(* IEC 61131-3 sources: volt/packages/volt-lsp-iec/test-corpus/pro2193/Device/Plc Logic/Application/99 Library/Function Blocks/Timers, 6 files *)

(* ---- BTOF.pou ---- *)
// Brink-TOF
{attribute 'no_explicit_call' := 'Do not call the body of BTOF directly! Use methods like Set to interact with this FB'}
{attribute 'monitoring_display' := 'TOF1.ET'}
FUNCTION_BLOCK FINAL BTOF
VAR
	TOF1		: Standard.TOF;
END_VAR

// Use methods to interact with the FB.

%LANGUAGE ST

END_FUNCTION_BLOCK

// Reset the timer.
METHOD PUBLIC Reset

%LANGUAGE ST
TOF1(IN := FALSE);

END_METHOD

// Set Brink timer
METHOD PUBLIC Set : BOOL
VAR_INPUT
	In	: BOOL;	// Starts timer with rising edge, stops timer with falling edge
	Pt	: REAL;	// Time to pass (in sec.), before Q is set
END_VAR

%LANGUAGE ST
TOF1(
	IN := In,
	PT := TO_TIME(Pt * 1000),
	Q  => ,
	ET => );

Set := TOF1.Q;

END_METHOD

// Monitor the output Q of the timer
{attribute 'monitoring':='call'}
PROPERTY PUBLIC Q : BOOL

GET
VAR
END_VAR

%LANGUAGE ST
Q := TOF1.Q;

END_GET
END_PROPERTY

(* ---- BTON.pou ---- *)
// Brink-TON
{attribute 'no_explicit_call' := 'Do not call the body of BTOF directly! Use methods like Set to interact with this FB'}
{attribute 'monitoring_display' := 'TON1.ET'}
FUNCTION_BLOCK FINAL BTON
VAR
	TON1		: Standard.TON;
END_VAR

// Use methods to interact with the FB.

%LANGUAGE ST

END_FUNCTION_BLOCK

// Reset the timer.
METHOD PUBLIC Reset

%LANGUAGE ST
TON1(IN := FALSE);

END_METHOD

// Set Brink timer
METHOD PUBLIC Set : BOOL
VAR_INPUT
	In	: BOOL;	// Starts timer with rising edge, stops timer with falling edge
	Pt	: REAL;	// Time to pass (in sec.), before Q is set
END_VAR

%LANGUAGE ST
TON1(
	IN := In,
	PT := TO_TIME(Pt * 1000),
	Q  => ,
	ET => );

Set := TON1.Q;

END_METHOD

// Monitor the output Q of the timer
{attribute 'monitoring':='call'}
PROPERTY PUBLIC Q : BOOL

GET
VAR
END_VAR

%LANGUAGE ST
Q := TON1.Q;

END_GET
END_PROPERTY

(* ---- MeasureTime.pou ---- *)
// Count time (in sec) how long an input is high/active. Counter resets when input is low.
{attribute 'no_explicit_call' := 'Do not call the body of MeasureModuleTime directly! Use methods to interact with this FB'}
{attribute 'hide_all_locals'}
{attribute 'monitoring_display' := 'rStoredTime'}
FUNCTION_BLOCK MeasureTime
VAR_OUTPUT
	rStoredTimeMax	: REAL;
END_VAR
VAR
	TON1			: Standard.TON;
	rStoredTime		: REAL;		// Dynamic - The currently elapsed time while measuring. Resets when a new measurement starts.
END_VAR

%LANGUAGE ST

END_FUNCTION_BLOCK

// Measure the time how long a condition is true.
METHOD PUBLIC Measure : REAL
VAR_INPUT
	In	: BOOL;	// Measure the time the input remains high
END_VAR

%LANGUAGE ST
IF (In XOR TON1.IN)				// Triggers the first cycle In is true, and the first cycle In is false. Give output.
OR (In AND TON1.ET > T#1S)		// Output will start running when timer has been running for more than 1 sec.
THEN
	rStoredTime		:= TO_REAL(TON1.ET) / 1000;
END_IF

IF NOT In AND TON1.IN THEN
	rStoredTimeMax	:= TO_REAL(TON1.ET) / 1000;
END_IF

TON1(
	IN := In,
	PT := GVL_Constants.TimeLongest,
	Q  => ,
	ET => );

Measure := rStoredTime;			// Give the output

END_METHOD

// Get elapsed time value
{attribute 'monitoring':='call'}
PROPERTY PUBLIC ElapsedTime : REAL

GET
VAR
END_VAR

%LANGUAGE ST
ElapsedTime := rStoredTime;

END_GET
END_PROPERTY

(* ---- ONTIME.pou ---- *)
// ONTIME measures the total time that a signal is active
{attribute 'monitoring_display' := 'udiSeconds'}
FUNCTION_BLOCK ONTIME
VAR_INPUT
	In			: BOOL;
END_VAR
VAR
	Last		: CAA.TICK;
	edge		: BOOL;
	udiMs		: UDINT;

	udiSeconds	: UDINT;	// Non-resetting ever-increasing time In is high
	udiCycles	: UDINT;	// Number of times the input switched on
	refSeconds	: REFERENCE TO UDINT REF= udiSeconds;
	refCycles	: REFERENCE TO UDINT REF= udiCycles;
END_VAR

%LANGUAGE ST
Initialize();

IF In THEN
	udiMs			:= udiMs + (TICKU.GetElapsedTimeInUSec(Last) / 1000);	// Add the elapsed milliseconds since last cycle

	IF udiMs >= 1000 THEN		// Check if a second has elapsed
		refSeconds	:= refSeconds + 1;
		udiMs		:= udiMs - 1000;
	END_IF

	refCycles		:= refCycles + TO_UDINT(NOT edge);
END_IF

Last				:= TICKS.GetTick(FALSE);
edge				:= In;

END_FUNCTION_BLOCK

METHOD PRIVATE Initialize
VAR_INST
	{attribute 'init_on_onlchange' }
	xInitialized	: BOOL;
END_VAR

%LANGUAGE ST
IF xInitialized THEN
	RETURN;
END_IF

Last			:= TICKS.GetTick(FALSE);
udiMs			:= 0;

xInitialized	:= TRUE;

END_METHOD

METHOD PUBLIC Reset
VAR_INPUT
END_VAR

%LANGUAGE ST
refSeconds		:= 0;
refCycles		:= 0;

Last			:= TICKS.GetTick(FALSE);
udiMs			:= 0;

END_METHOD

METHOD PUBLIC SetExternalCyclesReference
VAR_INPUT
	Cycles	: REFERENCE TO UDINT;
END_VAR

// We often need to persist the ONTIME data, so the data retains their value after reboots.
// For example if we count how long a vacuumpump has been running.
// In that case we need to declare the data in the PersistentVars list
// Use this method to set a reference to that variable

// If this method is never used (or reference is set to NULL), data is counted internally in the FB.

%LANGUAGE ST
IF __ISVALIDREF(Cycles) THEN
	THIS^.refCycles		REF= Cycles;
ELSE
	THIS^.refCycles		REF= udiCycles;
END_IF

END_METHOD

METHOD PUBLIC SetExternalSecondsReference
VAR_INPUT
	Seconds	: REFERENCE TO UDINT;
END_VAR

// We often need to persist the ONTIME data, so the data retains their value after reboots.
// For example if we count how long a vacuumpump has been running.
// In that case we need to declare the data in the PersistentVars list
// Use this method to set a reference to that variable

// If this method is never used (or reference is set to NULL), data is counted internally in the FB.

%LANGUAGE ST
IF __ISVALIDREF(Seconds) THEN
	THIS^.refSeconds	REF= Seconds;
ELSE
	THIS^.refSeconds	REF= udiSeconds;
END_IF

END_METHOD

{attribute 'monitoring':='call'}
PROPERTY PUBLIC AsReal : REAL

GET
VAR
END_VAR

%LANGUAGE ST
AsReal := TO_REAL(refSeconds) + TO_REAL(udiMs) / 1000;

END_GET
END_PROPERTY

{attribute 'monitoring':='call'}
PROPERTY PUBLIC AsTime : TIME

GET
VAR
END_VAR

%LANGUAGE ST
AsTime := TO_TIME(refSeconds * 1000 + udiMs);

END_GET
END_PROPERTY

{attribute 'monitoring':='call'}
PROPERTY PUBLIC Cycles : ULINT

GET
VAR
END_VAR

%LANGUAGE ST
Cycles := refCycles;

END_GET
END_PROPERTY

{attribute 'monitoring':='call'}
PROPERTY PUBLIC InSeconds : ULINT

GET
VAR
END_VAR

%LANGUAGE ST
InSeconds := refSeconds;

END_GET
END_PROPERTY

(* ---- SignalTimeoutFB.pou ---- *)
// This FB compares the input signal to the expected value, and will throw an alarm when the result is not as expected within a given time.
// The GetValue method returns the input value, and starts the timeout timer.
// The timer runs as long as the GetValue is called in every successive PLC cycle, the first cycle in which it is not called, it will reset the timer.
FUNCTION_BLOCK SignalTimeoutFB
VAR_INPUT
	input		: BOOL;			// Input signal
	timeOut		: REAL := 5;	// Timout for alarm  (default: 5s)
END_VAR
VAR_OUTPUT
	alarmActive	: BOOL;			// Input is not equal to Expected within the given timeout
END_VAR
VAR
	requested	: BOOL;			// Toggle bit for detecting every GetValue call
	timer		: BTON;			// Alarm timer
END_VAR

%LANGUAGE ST
IF NOT requested THEN
	timer.Reset();
	alarmActive := FALSE;
END_IF

requested := FALSE;

END_FUNCTION_BLOCK

// Starts the timeout timer, and returns the input signal
METHOD GetValue : BOOL
VAR_INPUT
	expected : BOOL;
END_VAR

%LANGUAGE ST
alarmActive	:= timer.Set(In := input <> expected, Pt := timeOut);
requested	:= TRUE;
GetValue	:= input;

END_METHOD

(* ---- StopwatchFB.pou ---- *)
// Measure precise durations [µs]. Use to debug code and check how long code needs to run.
// Also use Monitor() method to measure duration of booleans
{attribute 'no_explicit_call' := 'Do not call the body of StopwatchFB directly! Use methods to interact with this FB'}
{attribute 'monitoring_display' := 'actTime'}
{attribute 'symbol' := 'none'}
FUNCTION_BLOCK PUBLIC StopwatchFB
EXTENDS MonitoringAddLogBase
VAR
	ltStart		: LTIME;
END_VAR
VAR_OUTPUT
	actTime		: UDINT;	// UDINT storing microseconds can represent roughly 4,295 seconds or 71,5 minutes before it overflows!
	minTime		: UDINT;
	maxTime		: UDINT;
END_VAR

%LANGUAGE ST

END_FUNCTION_BLOCK

// Returns measurement [µs]
METHOD PUBLIC End : UDINT

%LANGUAGE ST
IF TO_UDINT(ltStart) = 0 THEN
	RETURN;
END_IF

actTime		:= TO_UDINT(LTIME() - ltStart) / 1000;
minTime		:= SEL(minTime <> 0, actTime, MIN(minTime, actTime));
maxTime		:= SEL(maxTime <> 0, actTime, MAX(maxTime, actTime));
End			:= actTime;

CallAddLogLREAL(TO_LREAL(actTime) / 1_000_000);	// Log time in sec.

END_METHOD

// Measure the time [µs] that a signal is active, and outputs that time when the signal deactivates.
METHOD PUBLIC Monitor : UDINT // [µs]
VAR_INPUT
	in					: BOOL;
END_VAR
VAR_INST
	last				: BOOL;
END_VAR

%LANGUAGE ST
IF in XOR last THEN
	IF in THEN
		Start();
	ELSE
		End();
	END_IF
END_IF
last	:= in;
Monitor := actTime;

END_METHOD

// Resets minimum and maximum values
METHOD PUBLIC Reset

%LANGUAGE ST
actTime		:= 0;
minTime		:= 0;
maxTime		:= 0;

END_METHOD

// Starts measurement
METHOD PUBLIC Start

%LANGUAGE ST
ltStart := LTIME();

END_METHOD
